PROGRAM MAIN
VAR
	
	//Pulsador AT %I*: BOOL;
	//Lampara AT %Q*: BOOL;
	
	Selector_modo_manual AT %I*: BOOL;
	
	test_pieza: FB_Bloque;

END_VAR

IF NOT Selector_modo_manual THEN
test_pieza();
END_IF

END_PROGRAM

(* stored: Version 1.1.0.1, ProductVersion 3.1.4024.12
   POU MAIN: Id {f8efd561-8056-4b52-b326-5a4dfa7df24d}, SpecialFunc None *)
